INTERFACE ITF_PackMLV2

METHOD Abort : BOOL
VAR_INPUT
END_VAR
END_METHOD

METHOD Clear : BOOL
VAR_INPUT
END_VAR
END_METHOD

{warning 'add method implementation '}
METHOD FB_init : BOOL
VAR_INPUT
	(* if TRUE, the retain variables are initialized (warm start / cold start)*)
	bInitRetains	: BOOL;
	(* if TRUE, the instance afterwards gets moved into the copy code (online change)*)
	bInCopyCode	: BOOL;
END_VAR
END_METHOD

METHOD Hold : BOOL
VAR_INPUT
END_VAR
END_METHOD

METHOD Reset : BOOL
VAR_INPUT
END_VAR
END_METHOD

METHOD Start : BOOL
VAR_INPUT
END_VAR
END_METHOD

PROPERTY State : E_State_PackML
GET
END_GET
END_PROPERTY

METHOD Stop : BOOL
VAR_INPUT
END_VAR
END_METHOD

METHOD Suspend : BOOL
VAR_INPUT
END_VAR
END_METHOD

METHOD Unhold : BOOL
VAR_INPUT
END_VAR
END_METHOD

METHOD Unsuspend : BOOL
VAR_INPUT
END_VAR
END_METHOD

METHOD ZeroAllVar : BOOL
VAR_INPUT
END_VAR
END_METHOD

END_INTERFACE

(* stored: Version 1.1.0.1, ProductVersion 3.1.4024.12
   Itf ITF_PackMLV2: Id {f36d244c-592b-4934-bf10-34d2733c2b69}
   Folder Methods: Id {1415d138-6fce-433a-a6e3-630eafd51c12}
   Folder Properties: Id {7331e99e-4d30-4727-9f07-4fec1ff35076}
   Method Abort: Id {258eb838-12f8-418f-a21b-10e12e6fe1ff}
   Method Clear: Id {90f5b295-1a23-424a-9105-0655e4199011}
   Method FB_init: Id {99d1fb55-0fe0-444a-9eb4-e16e1f22f624}
   Method Hold: Id {b6497211-0bbc-4ba8-b83f-bbbef2cd7d19}
   Method Reset: Id {2ebbb344-22d5-4b5b-b428-fd54e96fc351}
   Method Start: Id {3441e2e5-c47a-43a8-a154-f1c799d55473}
   Property State: Id {1617ead2-2391-4ad5-b863-b8547dca6453}
   Get Get: Id {0ee5baa0-eafa-4b9a-ab55-8e84fc3668b7}
   Method Stop: Id {955fd5f7-1d40-4d66-80f4-261e4a67bd86}
   Method Suspend: Id {7feca0df-c7da-45f7-ba8c-25f3d6f33e76}
   Method Unhold: Id {27293311-4c3b-48d9-be55-26355fdc71e5}
   Method Unsuspend: Id {438438d9-f343-4545-aa33-1f9c9a4d04fa}
   Method ZeroAllVar: Id {45f42221-f955-45c3-8ea2-5cc6a747c668} *)
